# EPICS autosave request: motorSimApp/Db/motorSim_settings.req
file "basic_motor_settings.req", P=test:,M=m1
file "basic_motor_settings.req", P=test:,M=m2
file "basic_motor_settings.req", P=test:,M=m3
file "basic_motor_settings.req", P=test:,M=m4
file "basic_motor_settings.req", P=test:,M=m5
file "basic_motor_settings.req", P=test:,M=m6
